PROGRAM MAIN
VAR
	
	tonCopy :	TON;
END_VAR


tonCopy(in:=NOT(tonCopy.Q), PT:=T#900MS);

IF tonCopy.Q THEN
	POU_copyXmeasXmv();
END_IF

END_PROGRAM

(* stored: Version 1.1.0.1, ProductVersion 3.1.4024.11
   POU MAIN: Id {7ebce504-5f6f-4ed6-935e-d786a7755d0f}, SpecialFunc None *)
